FUNCTION_BLOCK NAND_BOOL (* Boolean NOT_AND *)
  (* Standard: 61131-3 *)
  (* Version 0.0, 2006-09-19, JHC, Holobloc Inc, Derived from AND_BOOL. *)
  (* Compiler header: package fb.rt.plc.bits; *)
  (* Compiler classdef: (!( i1 && i2 )) *)
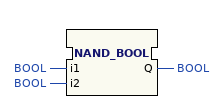
  VAR_INPUT
    i1 : BOOL;
    i2 : BOOL;
  END_VAR
  VAR_OUTPUT
    Q : BOOL;
  END_VAR
END_FUNCTION_BLOCK
